Universal Robots PolyScope program: demo sleeve flush cw.urp

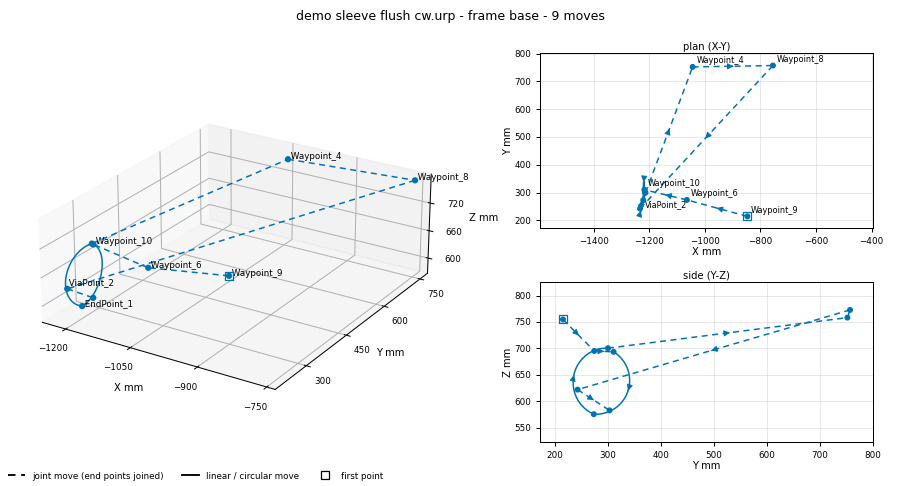
[picture p0: tool path of demo sleeve flush cw.urp in frame base, 9 of 11 moves have a stored position in this frame; points joined in program order, loops and branches not executed]
Program demo sleeve flush cw (installation=default directory=/programs createdIn=5.21.3 lastSavedIn=5.21.3 robotSerialNumber=20246801938)
Calibrated DH parameters: a=[-0.000071, -0.790281, -0.600694, 0.000061, -0.000039, 0]; d=[0.236272, 604.465945, 132.116513, -736.382239, 0.159268, 0.154005]; alpha=[1.570254, -0.000567, 0.000559, 1.571709, -1.56999, 0]; deltaTheta=[0, -0.409357, 7.293326, -0.600784, -0.000001, -0.000001]
InitVariablesNode
Robot Program (runOnlyOnce=false)
  MoveJ speed 60 deg/s, acceleration 80 deg/s^2 (useActiveTCP=true optimoveEnabled=false optiMoveSpeed=0.3 optiMoveAcceleration=0.09) feature=Base
    SuppressedNode
      Waypoint Waypoint_3: TCP in base x=-912.453 y=673.518 z=718.985 mm, rx=-0.4706 ry=-1.9428 rz=0.4955 rad; joints [-63.285, -68.284, 110.161, 88.985, -83.541, -118.353] deg; TCP offset x=-9.5 y=-328 z=105.73 mm, rx=1.2092 ry=-1.2092 rz=1.2092 rad
    SuppressedNode
      Waypoint Waypoint_4: TCP in base x=-1043.534 y=752.126 z=758.241 mm, rx=-0.4498 ry=-2.3257 rz=-0.2665 rad; joints [-53.991, -67.414, 94.218, 102.936, -66.691, -159.337] deg
    Waypoint Waypoint_9: TCP in base x=-846.524 y=214.492 z=754.78 mm, rx=0.075 ry=-1.6382 rz=-0.3957 rad; joints [-44.538, -78.526, 126.302, -324.644, -73.702, -146.265] deg
    Waypoint Waypoint_6: TCP in base x=-1064.157 y=273.628 z=695.243 mm, rx=-2.0108 ry=-0.057 rz=2.2447 rad; joints [-33.712, -99.226, 114.776, -114.381, -92.359, -30.249] deg
  MoveJ speed 60 deg/s, acceleration 80 deg/s^2 (useActiveTCP=true optimoveEnabled=false optiMoveSpeed=0.3 optiMoveAcceleration=0.09) feature=Base
    SuppressedNode
      Waypoint Waypoint_1: TCP in base x=-1152.594 y=814.679 z=699.964 mm, rx=0.098 ry=-2.3843 rz=-0.4483 rad; joints [-56.525, -54.403, 73.307, 93.455, -42.841, -145.624] deg
    SuppressedNode
      Waypoint Waypoint_5: TCP in base x=-1149.758 y=814.958 z=702.794 mm, rx=-0.0472 ry=-2.3472 rz=-0.7271 rad; joints [-53.278, -57.004, 80.845, -264.711, -44.526, -166.31] deg
    SuppressedNode
      Waypoint Waypoint_7: TCP in base x=-1212.936 y=299.576 z=700.501 mm, rx=0.0471 ry=-1.5574 rz=-0.1368 rad; joints [-31.134, -66.409, 121.876, -149.38, 84.433, 28.033] deg
    Waypoint Waypoint_10: TCP in base x=-1217.118 y=310.24 z=693.595 mm, rx=-0.1891 ry=-1.666 rz=-0.1324 rad; joints [-27.214, -71.949, 123.303, -135.263, -270.241, 15.61] deg
  MoveP speed 10 mm/s, acceleration 1200 mm/s^2 (blendRadius=0.025 useActiveTCP=true optimoveEnabled=false optiMoveSpeed=0.3 optiMoveAcceleration=0.09) feature=Base
    CircleMove (OrientationMode=FIXED)
      Waypoint ViaPoint_1: TCP in base x=-1219.861 y=338.76 z=624.282 mm, rx=-1.5212 ry=-0.9663 rz=1.2658 rad; joints [-15.001, -79.342, 112.744, -139.734, -163.22, -20.907] deg
      Waypoint EndPoint_1: TCP in base x=-1221.187 y=272.785 z=575.704 mm, rx=-2.2635 ry=0.1661 rz=2.1342 rad; joints [-28.617, -84.967, 103.188, -103.722, -88.538, -23.283] deg
    CircleMove (OrientationMode=FIXED)
      Waypoint ViaPoint_2: motionParameters(blendRadius=0); TCP in base x=-1230.114 y=233.667 z=633.743 mm, rx=1.3046 ry=-1.4594 rz=-1.7128 rad; joints [-34.044, -85.948, 110.193, -88.024, -21.173, -24.678] deg
      Waypoint Waypoint_7: motionParameters(blendRadius=0); TCP in base x=-1212.936 y=299.576 z=700.501 mm, rx=0.0471 ry=-1.5574 rz=-0.1368 rad; joints [-31.134, -66.409, 121.876, -149.38, 84.433, 28.033] deg
  MoveJ speed 60 deg/s, acceleration 80 deg/s^2 (useActiveTCP=true optimoveEnabled=false optiMoveSpeed=0.3 optiMoveAcceleration=0.09) feature=Base
    SuppressedNode
      Waypoint Waypoint_2: TCP in base x=-917.75 y=830.261 z=524.512 mm, rx=-1.543 ry=-0.8444 rz=1.9881 rad; joints [-66.08, -72.484, 118.808, 175.962, -93.351, -73.55] deg
    Waypoint Waypoint_4: TCP in base x=-1043.534 y=752.126 z=758.241 mm, rx=-0.4498 ry=-2.3257 rz=-0.2665 rad; joints [-53.991, -67.414, 94.218, 102.936, -66.691, -159.337] deg
    Waypoint Waypoint_8: TCP in base x=-754.583 y=757.082 z=772.781 mm, rx=-0.4498 ry=-2.3257 rz=-0.2665 rad; joints [-73.782, -79.343, 107.572, 92.439, -55.198, -140.846] deg
  MoveJ speed 60 deg/s, acceleration 80 deg/s^2 (useActiveTCP=true optimoveEnabled=false optiMoveSpeed=0.3 optiMoveAcceleration=0.09) feature=Base
    Waypoint Waypoint_11: TCP in base x=-1232.726 y=242.18 z=622.16 mm, rx=-1.2679 ry=-1.1266 rz=1.051 rad; joints [-8.14, -73.065, 115.912, -155.85, -182.636, -24.18] deg
    Waypoint Waypoint_12: TCP in base x=-1215.592 y=302.474 z=582.981 mm, rx=-0.1781 ry=-1.5815 rz=-0.0746 rad; joints [-26.703, -61.115, 124.943, -151.661, -266.873, 17.546] deg
